// SIMATIC S7-200 project (STEP 7-Micro/WIN), CPU 224 REL 02.01

SYMBOL_TABLE USER1
Gain             600
Ut2              VB1
Ut               QW1
Td               250
Et               VW1      // Check
Heater           Q0.0
END_SYMBOL_TABLE

ORGANIZATION_BLOCK MAIN:OB1
TITLE=PROGRAM COMMENTS
VAR
Et:INT;	// LW0 error
END_VAR
BEGIN
Network 1 // Network Title
// Network Comment
// (network saved uncompiled; FBD cells follow)
// row 0: c1 [SUB_I ]  c4 [MUL_I ]  c7 [ENCO ]  c10 [DECO ]
// row 1: c1 [ EN:=I0.0, IN1:=AIW8, IN2:=Td, ENO=>power, OUT=>#Et:LW0]  c2 --  c3 --  c4 [ EN:=power@row1, IN1:=#Et:LW0, IN2:=Gain, ENO=>power, OUT=>Ut:QW1]  c5 --  c6 --  c7 [ EN:=power@row1, IN:=Ut:QW1, ENO=>power, OUT=>Ut2:VB1]  c8 --  c9 --  c10 [ EN:=power@row1, IN:=Ut2:VB1, ENO=>V?0, OUT=>AQW0]
// row 2: c1 [box]  c4 [box]  c7 [box]  c10 [box]
// row 3: c1 [box]  c4 [box]
Network 2
LDW<   AIW8, Td
=      Heater:Q0.0
END_ORGANIZATION_BLOCK
